//TxRxBuffer provided by ComPortEL6x22BEasyConnect FB to be sued by ComPortDeviceCom_SendRecBytes/String
FUNCTION_BLOCK ComPortDeviceCom_BufferHandle
VAR CONSTANT										
END_VAR
VAR_INPUT
	TXBuffer												: 	COMbuffer ;	
	RXBuffer												: 	COMbuffer ;
END_VAR		
VAR_OUTPUT
END_VAR
VAR_IN_OUT
END_VAR
VAR_OUTPUT
END_VAR
VAR
	ClearComBuf												:	ClearComBuffer;
END_VAR

	(* RS232 Device Com										 *)
	(*********************************************************)

METHOD PUBLIC clear : BOOL
VAR_INPUT
END_VAR
ClearComBuf(Buffer := RXBuffer);
ClearComBuf(Buffer := TXBuffer);
Clear 										:= TRUE;
END_METHOD

METHOD PUBLIC clearRxBuffer : BOOL
VAR_INPUT
END_VAR
ClearComBuf(Buffer := RXBuffer);
ClearRxBuffer 									:= TRUE;
END_METHOD

METHOD PUBLIC clearTxBuffer : BOOL
VAR_INPUT
END_VAR

ClearComBuf(Buffer := TXBuffer);
ClearTxBuffer 										:= TRUE;
END_METHOD

END_FUNCTION_BLOCK

(* stored: Version 1.1.0.1, ProductVersion 3.1.4024.13
   POU ComPortDeviceCom_BufferHandle: Id {06d44f9f-de92-46a6-b54b-5d50d34635bf}, SpecialFunc None
   Method clear: Id {8d873f97-1b9d-48f9-91c0-6505919965ec}
   Method clearRxBuffer: Id {57e27e13-6568-4040-81b5-f2610cce5d43}
   Method clearTxBuffer: Id {2dd28c3b-7bc4-4aaf-be15-9db1c4c71ad8} *)
